RoboDK station: envolope-station.rdk

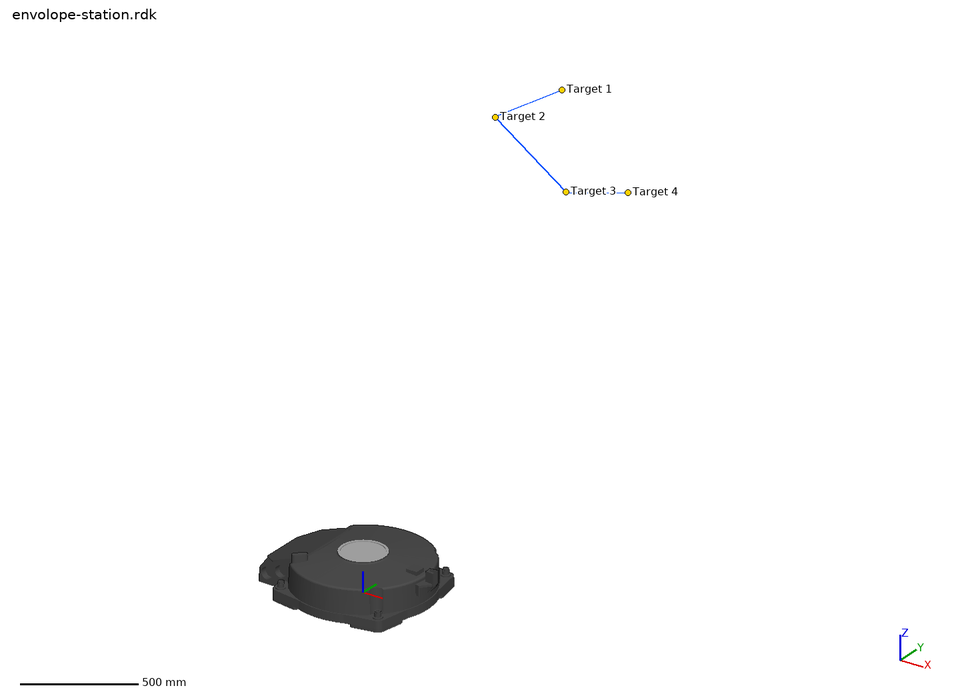
[picture v0: the station drawn from its stored meshes, robots at their saved joint values, targets as dots, program paths as lines]
Station envolope-station (saved by RoboDK 5.7.4). Poses are relative to the parent item; angles as X-Y-Z fixed-axis rotations.
  - frame ABB IRB 580/12S Base at (0, 0, 0) mm
    - robot ABB IRB 580/12S: 6 axes, payload 12 kg, reach 2200 mm, repeatability 0.3 mm, weight 630 kg
        joint limits [-150, -70, -145, -360, -360, -720] to [150, 75, 145, 360, 360, 720]; home [0, 0, 0, 0, 0, 0]; saved at [79.62, -15.02, -23.42, 357.92, -41.53, -38.08]
    - target Target 1 (Cartesian target) at (151.38, 1247.14, 1902.22) mm, rotated rx -75.77 ry 7.65 rz 14.35 deg; joints [79.62, 17.98, -23.42, 357.92, -41.53, -38.08] of ABB IRB 580/12S
    - target Target 2 (Cartesian target) at (79.77, 856.16, 1912.49) mm, rotated rx -75.77 ry 7.65 rz 14.35 deg; joints [79.62, -15.02, -23.42, 357.92, -41.53, -38.08] of ABB IRB 580/12S
    - target Target 3 (Cartesian target) at (741.36, 435.61, 1912.49) mm, rotated rx -75.77 ry 7.65 rz -39.89 deg; joints [25.38, -15.02, -23.42, 357.92, -41.53, -38.08] of ABB IRB 580/12S
    - target Target 4 (Cartesian target) at (981.02, 549.3, 1931.37) mm, rotated rx -75.77 ry 7.65 rz -39.89 deg; joints [25.38, 6.88, -23.42, 357.92, -41.53, -38.08] of ABB IRB 580/12S
  - program Prog1 (5 instructions, listed below)
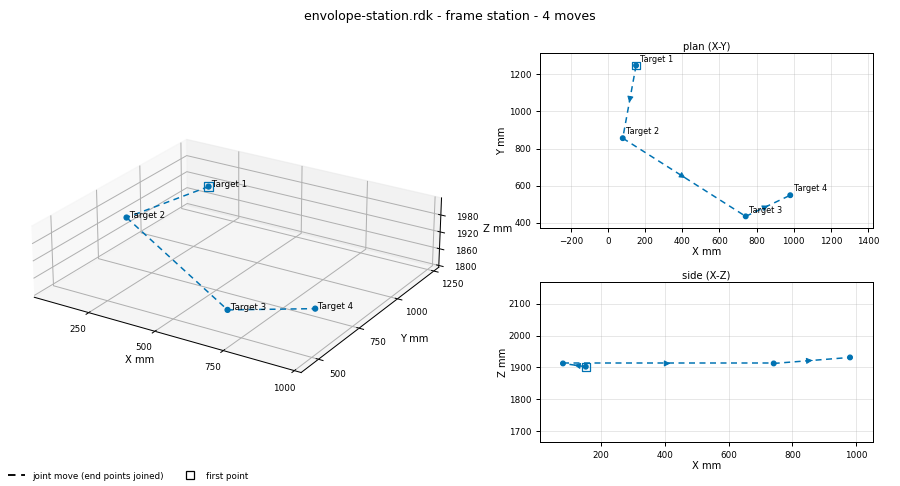
[picture p0: tool path of envolope-station.rdk in frame station, 4 of 4 moves have a stored position in this frame; points joined in program order, loops and branches not executed]

--- program Prog1 (robot ABB IRB 580/12S) ---
  Set Ref.: ABB IRB 580/12S Base
  MoveJ (Target 1)
  MoveJ (Target 2)
  MoveJ (Target 3)
  MoveJ (Target 4)
